{attribute 'qualified_only'}
VAR_GLOBAL
	uniDI : uni_InputModule;
END_VAR

(* stored: Version 1.1.0.1, ProductVersion 3.1.4024.13
   GVL GVL_Input: Id {415bfdd1-81e5-447f-a7d5-262cb553aaae} *)
